(*
Nazwa:			E_MachineState
Opis:			Stan masyzny
Wersja:			v0.1
Data:			2018-10-10
Autor:			TW,DP
Urzadzenia:		
Konfiguracja:	
Info:
*)

//{attribute 'strict'}
//{attribute 'qualified_only'}
TYPE E_MachineState :
(
	eOn := 0, //Właczono
	ePower := 1, //Zasilanie
	eIdle := 2,	//Inicjacja
	eWaitingForPositioning := 4, //Czekanie na bazowanie
	ePositioning := 5, //Bazowanie
	eReady := 6, //Gotowa
	eServiceMode := 7, //Tryb Serwisowy
	eEnginesOn := 8, //Silniki włączone
	eCycleStarting := 9, //Start cyklu
	eCycleOn := 10, //Praca
	eStopping := 11, //Zatrzymywanie
	eConfectionStart := 12, //Start konfekcji
	eConfectionEnd := 13, //Stop konfekcji
	eHardError := 20, //Bład safety
	eSoftError := 21, //Bład
	eAfterError := 22, //Przywracanie po błedzie
	eReset := 30 //Resetowanie
);
END_TYPE

(* stored: Version 1.1.0.1, ProductVersion 3.1.4026.13, FileIdentifier cb3321f269e5375dd86ce391cdd79640be8af990, FileSignature 139232c4bbb010b4660b23def8088c9bd78e686d5c405276a8ea67fcdbb6a13874346da6e12771994a2bf7f73d7807b9a28a1de711ab0ba9fd3f0c03cfe8e9fe5b1b49a0a2b539c55325903fc558fb20fd3337913cf00ef1bbec002483e51bd0b2028f0c46b7fbfd37cc5d9991148b975f4eda2ee7198dce3507682cd637df28690bc5f1b8dbfcd80b1877d7414bbd8e8eabe2ed97ee78c41b10c3b41eb05e0c99f932694b83c2b13a15c3fe56ad39849083b6a990342d15e4e85a35648430d777f6ec11992a0ff493ec6e6a588d55222394204168e55e8a4e107a408c29afa772a7becc7c23f376960d4a8713764af1e4534609eb7d685b0f70430ca847e524
   DUT E_MachineState: Id {ab892143-d035-4f22-bf30-d53fc0d5f0ff} *)
